Staubli VAL3: getPalletPos.pgx

public program getPalletPos(string x_sItem, num& x_nIndex[])
  local num i
  local string l_sName
  local num l_nPos
  local num l_nSize
begin
  // init the index
  x_nIndex=-1
  // scan it
  if isDefined(pt:tTraj[x_sItem])
    x_nIndex=pt:tTraj[x_sItem].nIndex
    //
  endIf
end
